INTERFACE interface3

METHOD itf_metodo : BOOL
VAR_INPUT
END_VAR
END_METHOD

PROPERTY itf_propiedad : real
GET
END_GET
SET
END_SET
END_PROPERTY

END_INTERFACE

(* stored: Version 1.1.0.1, ProductVersion 3.1.4024.12
   Itf interface3: Id {605f177d-96c4-4a3f-87fc-212bc8e919d8}
   Method itf_metodo: Id {ba7026e5-04c8-451b-87ee-1522cd16d8f3}
   Property itf_propiedad: Id {276581cf-9564-47cb-bd95-776e8a060b0d}
   Get Get: Id {8b201810-01ee-44e6-9f6d-b0ed3f5b4e04}
   Set Set: Id {a572f6dc-dd26-4646-8522-e4407f90c4fa} *)
